// TIA Portal V18 export
// export: Created 2026-06-08T06:16:14.4955932Z, ExportSetting WithDefaults, DisplayName Totally Integrated Automation Portal, DisplayVersion V18, DisplayName TIA Portal Openness, DisplayVersion V18, DisplayName TIA Portal Version Control Interface, DisplayVersion V18, DisplayName STEP 7 Professional, DisplayVersion V18, DisplayName STEP 7 Safety, DisplayVersion V18, DisplayName WinCC Professional, DisplayVersion V18
FUNCTION "FC_Bon_Chua_Loc" : Void   // FC30, LAD
{ S7_Optimized_Access := 'TRUE' }
VERSION : 0.1
// stored: AutoNumber true, IsIECCheckEnabled false, SetENOAutomatically false, UDAEnableTagReadback false
BEGIN

REGION Network 1: Gated HMI AI_LSH3310_Pheu_Cao qua Sim Mode
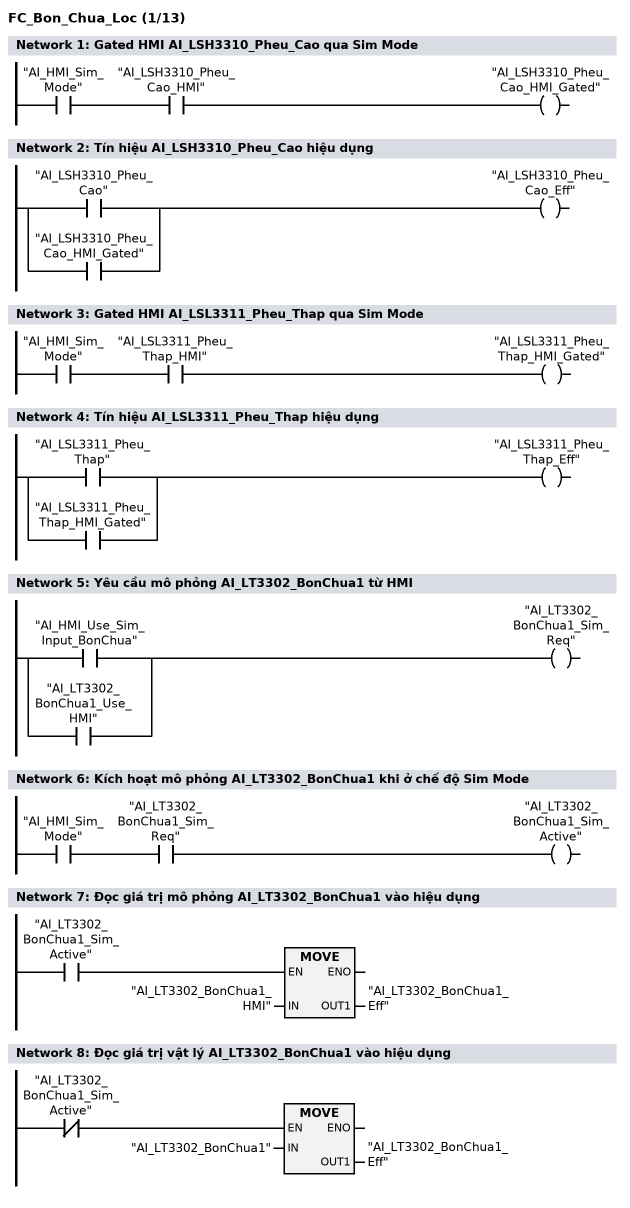
   RUNG wire#powerrail
      Contact( "AI_HMI_Sim_Mode" )
      Contact( "AI_LSH3310_Pheu_Cao_HMI" )
      Coil( "AI_LSH3310_Pheu_Cao_HMI_Gated" )
   END_RUNG
   // the same network as SCL:
   "AI_LSH3310_Pheu_Cao_HMI_Gated" := "AI_HMI_Sim_Mode" AND "AI_LSH3310_Pheu_Cao_HMI";
END_REGION

REGION Network 2: Tín hiệu AI_LSH3310_Pheu_Cao hiệu dụng
   RUNG wire#powerrail
      Contact( "AI_LSH3310_Pheu_Cao" )
      wire#w1
      Coil( "AI_LSH3310_Pheu_Cao_Eff" )
   END_RUNG
   RUNG wire#powerrail
      Contact( "AI_LSH3310_Pheu_Cao_HMI_Gated" )
   END_RUNG wire#w1
   // the same network as SCL:
   "AI_LSH3310_Pheu_Cao_Eff" := "AI_LSH3310_Pheu_Cao" OR "AI_LSH3310_Pheu_Cao_HMI_Gated";
END_REGION

REGION Network 3: Gated HMI AI_LSL3311_Pheu_Thap qua Sim Mode
   RUNG wire#powerrail
      Contact( "AI_HMI_Sim_Mode" )
      Contact( "AI_LSL3311_Pheu_Thap_HMI" )
      Coil( "AI_LSL3311_Pheu_Thap_HMI_Gated" )
   END_RUNG
   // the same network as SCL:
   "AI_LSL3311_Pheu_Thap_HMI_Gated" := "AI_HMI_Sim_Mode" AND "AI_LSL3311_Pheu_Thap_HMI";
END_REGION

REGION Network 4: Tín hiệu AI_LSL3311_Pheu_Thap hiệu dụng
   RUNG wire#powerrail
      Contact( "AI_LSL3311_Pheu_Thap" )
      wire#w1
      Coil( "AI_LSL3311_Pheu_Thap_Eff" )
   END_RUNG
   RUNG wire#powerrail
      Contact( "AI_LSL3311_Pheu_Thap_HMI_Gated" )
   END_RUNG wire#w1
   // the same network as SCL:
   "AI_LSL3311_Pheu_Thap_Eff" := "AI_LSL3311_Pheu_Thap" OR "AI_LSL3311_Pheu_Thap_HMI_Gated";
END_REGION

REGION Network 5: Yêu cầu mô phỏng AI_LT3302_BonChua1 từ HMI
   RUNG wire#powerrail
      Contact( "AI_HMI_Use_Sim_Input_BonChua" )
      wire#w1
      Coil( "AI_LT3302_BonChua1_Sim_Req" )
   END_RUNG
   RUNG wire#powerrail
      Contact( "AI_LT3302_BonChua1_Use_HMI" )
   END_RUNG wire#w1
   // the same network as SCL:
   "AI_LT3302_BonChua1_Sim_Req" := "AI_HMI_Use_Sim_Input_BonChua" OR "AI_LT3302_BonChua1_Use_HMI";
END_REGION

REGION Network 6: Kích hoạt mô phỏng AI_LT3302_BonChua1 khi ở chế độ Sim Mode
   RUNG wire#powerrail
      Contact( "AI_HMI_Sim_Mode" )
      Contact( "AI_LT3302_BonChua1_Sim_Req" )
      Coil( "AI_LT3302_BonChua1_Sim_Active" )
   END_RUNG
   // the same network as SCL:
   "AI_LT3302_BonChua1_Sim_Active" := "AI_HMI_Sim_Mode" AND "AI_LT3302_BonChua1_Sim_Req";
END_REGION

REGION Network 7: Đọc giá trị mô phỏng AI_LT3302_BonChua1 vào hiệu dụng
   RUNG wire#powerrail
      Contact( "AI_LT3302_BonChua1_Sim_Active" )
      { S7_GenerateENO := "TRUE" } Move(in := "AI_LT3302_BonChua1_HMI", out1 => "AI_LT3302_BonChua1_Eff")
   END_RUNG
   // the same network as SCL:
   IF "AI_LT3302_BonChua1_Sim_Active" THEN "AI_LT3302_BonChua1_Eff" := "AI_LT3302_BonChua1_HMI"; END_IF;
END_REGION

REGION Network 8: Đọc giá trị vật lý AI_LT3302_BonChua1 vào hiệu dụng
   RUNG wire#powerrail
      I_Contact( "AI_LT3302_BonChua1_Sim_Active" )
      { S7_GenerateENO := "TRUE" } Move(in := "AI_LT3302_BonChua1", out1 => "AI_LT3302_BonChua1_Eff")
   END_RUNG
   // the same network as SCL:
   IF NOT "AI_LT3302_BonChua1_Sim_Active" THEN "AI_LT3302_BonChua1_Eff" := "AI_LT3302_BonChua1"; END_IF;
END_REGION

REGION Network 9: Yêu cầu mô phỏng AI_TT3301_BonChua1 từ HMI
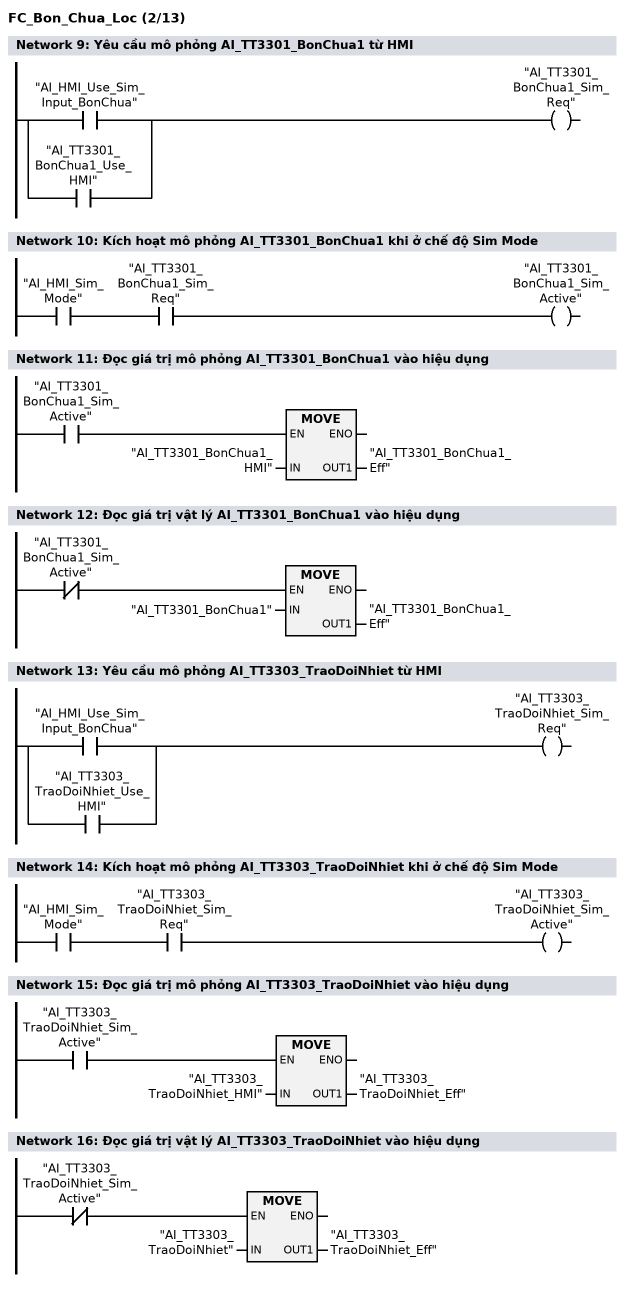
   RUNG wire#powerrail
      Contact( "AI_HMI_Use_Sim_Input_BonChua" )
      wire#w1
      Coil( "AI_TT3301_BonChua1_Sim_Req" )
   END_RUNG
   RUNG wire#powerrail
      Contact( "AI_TT3301_BonChua1_Use_HMI" )
   END_RUNG wire#w1
   // the same network as SCL:
   "AI_TT3301_BonChua1_Sim_Req" := "AI_HMI_Use_Sim_Input_BonChua" OR "AI_TT3301_BonChua1_Use_HMI";
END_REGION

REGION Network 10: Kích hoạt mô phỏng AI_TT3301_BonChua1 khi ở chế độ Sim Mode
   RUNG wire#powerrail
      Contact( "AI_HMI_Sim_Mode" )
      Contact( "AI_TT3301_BonChua1_Sim_Req" )
      Coil( "AI_TT3301_BonChua1_Sim_Active" )
   END_RUNG
   // the same network as SCL:
   "AI_TT3301_BonChua1_Sim_Active" := "AI_HMI_Sim_Mode" AND "AI_TT3301_BonChua1_Sim_Req";
END_REGION

REGION Network 11: Đọc giá trị mô phỏng AI_TT3301_BonChua1 vào hiệu dụng
   RUNG wire#powerrail
      Contact( "AI_TT3301_BonChua1_Sim_Active" )
      { S7_GenerateENO := "TRUE" } Move(in := "AI_TT3301_BonChua1_HMI", out1 => "AI_TT3301_BonChua1_Eff")
   END_RUNG
   // the same network as SCL:
   IF "AI_TT3301_BonChua1_Sim_Active" THEN "AI_TT3301_BonChua1_Eff" := "AI_TT3301_BonChua1_HMI"; END_IF;
END_REGION

REGION Network 12: Đọc giá trị vật lý AI_TT3301_BonChua1 vào hiệu dụng
   RUNG wire#powerrail
      I_Contact( "AI_TT3301_BonChua1_Sim_Active" )
      { S7_GenerateENO := "TRUE" } Move(in := "AI_TT3301_BonChua1", out1 => "AI_TT3301_BonChua1_Eff")
   END_RUNG
   // the same network as SCL:
   IF NOT "AI_TT3301_BonChua1_Sim_Active" THEN "AI_TT3301_BonChua1_Eff" := "AI_TT3301_BonChua1"; END_IF;
END_REGION

REGION Network 13: Yêu cầu mô phỏng AI_TT3303_TraoDoiNhiet từ HMI
   RUNG wire#powerrail
      Contact( "AI_HMI_Use_Sim_Input_BonChua" )
      wire#w1
      Coil( "AI_TT3303_TraoDoiNhiet_Sim_Req" )
   END_RUNG
   RUNG wire#powerrail
      Contact( "AI_TT3303_TraoDoiNhiet_Use_HMI" )
   END_RUNG wire#w1
   // the same network as SCL:
   "AI_TT3303_TraoDoiNhiet_Sim_Req" := "AI_HMI_Use_Sim_Input_BonChua" OR "AI_TT3303_TraoDoiNhiet_Use_HMI";
END_REGION

REGION Network 14: Kích hoạt mô phỏng AI_TT3303_TraoDoiNhiet khi ở chế độ Sim Mode
   RUNG wire#powerrail
      Contact( "AI_HMI_Sim_Mode" )
      Contact( "AI_TT3303_TraoDoiNhiet_Sim_Req" )
      Coil( "AI_TT3303_TraoDoiNhiet_Sim_Active" )
   END_RUNG
   // the same network as SCL:
   "AI_TT3303_TraoDoiNhiet_Sim_Active" := "AI_HMI_Sim_Mode" AND "AI_TT3303_TraoDoiNhiet_Sim_Req";
END_REGION

REGION Network 15: Đọc giá trị mô phỏng AI_TT3303_TraoDoiNhiet vào hiệu dụng
   RUNG wire#powerrail
      Contact( "AI_TT3303_TraoDoiNhiet_Sim_Active" )
      { S7_GenerateENO := "TRUE" } Move(in := "AI_TT3303_TraoDoiNhiet_HMI", out1 => "AI_TT3303_TraoDoiNhiet_Eff")
   END_RUNG
   // the same network as SCL:
   IF "AI_TT3303_TraoDoiNhiet_Sim_Active" THEN
       "AI_TT3303_TraoDoiNhiet_Eff" := "AI_TT3303_TraoDoiNhiet_HMI";
   END_IF;
END_REGION

REGION Network 16: Đọc giá trị vật lý AI_TT3303_TraoDoiNhiet vào hiệu dụng
   RUNG wire#powerrail
      I_Contact( "AI_TT3303_TraoDoiNhiet_Sim_Active" )
      { S7_GenerateENO := "TRUE" } Move(in := "AI_TT3303_TraoDoiNhiet", out1 => "AI_TT3303_TraoDoiNhiet_Eff")
   END_RUNG
   // the same network as SCL:
   IF NOT "AI_TT3303_TraoDoiNhiet_Sim_Active" THEN
       "AI_TT3303_TraoDoiNhiet_Eff" := "AI_TT3303_TraoDoiNhiet";
   END_IF;
END_REGION

REGION Network 17: Yêu cầu mô phỏng AI_LT3307_BonChua2 từ HMI
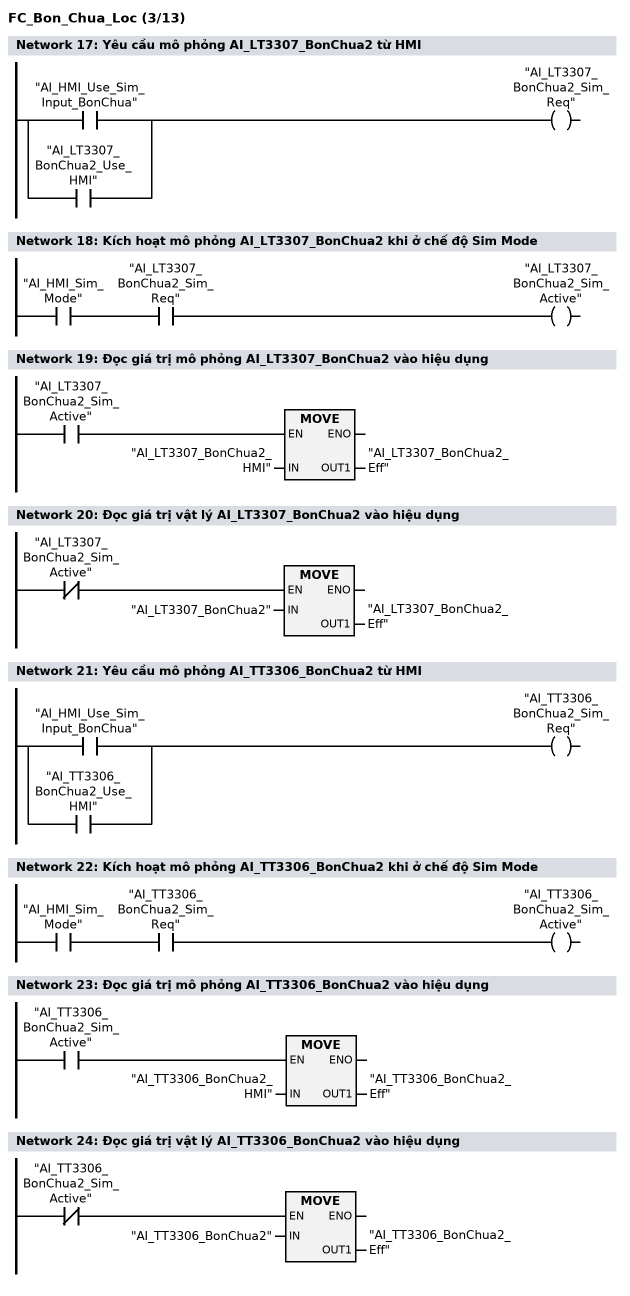
   RUNG wire#powerrail
      Contact( "AI_HMI_Use_Sim_Input_BonChua" )
      wire#w1
      Coil( "AI_LT3307_BonChua2_Sim_Req" )
   END_RUNG
   RUNG wire#powerrail
      Contact( "AI_LT3307_BonChua2_Use_HMI" )
   END_RUNG wire#w1
   // the same network as SCL:
   "AI_LT3307_BonChua2_Sim_Req" := "AI_HMI_Use_Sim_Input_BonChua" OR "AI_LT3307_BonChua2_Use_HMI";
END_REGION

REGION Network 18: Kích hoạt mô phỏng AI_LT3307_BonChua2 khi ở chế độ Sim Mode
   RUNG wire#powerrail
      Contact( "AI_HMI_Sim_Mode" )
      Contact( "AI_LT3307_BonChua2_Sim_Req" )
      Coil( "AI_LT3307_BonChua2_Sim_Active" )
   END_RUNG
   // the same network as SCL:
   "AI_LT3307_BonChua2_Sim_Active" := "AI_HMI_Sim_Mode" AND "AI_LT3307_BonChua2_Sim_Req";
END_REGION

REGION Network 19: Đọc giá trị mô phỏng AI_LT3307_BonChua2 vào hiệu dụng
   RUNG wire#powerrail
      Contact( "AI_LT3307_BonChua2_Sim_Active" )
      { S7_GenerateENO := "TRUE" } Move(in := "AI_LT3307_BonChua2_HMI", out1 => "AI_LT3307_BonChua2_Eff")
   END_RUNG
   // the same network as SCL:
   IF "AI_LT3307_BonChua2_Sim_Active" THEN "AI_LT3307_BonChua2_Eff" := "AI_LT3307_BonChua2_HMI"; END_IF;
END_REGION

REGION Network 20: Đọc giá trị vật lý AI_LT3307_BonChua2 vào hiệu dụng
   RUNG wire#powerrail
      I_Contact( "AI_LT3307_BonChua2_Sim_Active" )
      { S7_GenerateENO := "TRUE" } Move(in := "AI_LT3307_BonChua2", out1 => "AI_LT3307_BonChua2_Eff")
   END_RUNG
   // the same network as SCL:
   IF NOT "AI_LT3307_BonChua2_Sim_Active" THEN "AI_LT3307_BonChua2_Eff" := "AI_LT3307_BonChua2"; END_IF;
END_REGION

REGION Network 21: Yêu cầu mô phỏng AI_TT3306_BonChua2 từ HMI
   RUNG wire#powerrail
      Contact( "AI_HMI_Use_Sim_Input_BonChua" )
      wire#w1
      Coil( "AI_TT3306_BonChua2_Sim_Req" )
   END_RUNG
   RUNG wire#powerrail
      Contact( "AI_TT3306_BonChua2_Use_HMI" )
   END_RUNG wire#w1
   // the same network as SCL:
   "AI_TT3306_BonChua2_Sim_Req" := "AI_HMI_Use_Sim_Input_BonChua" OR "AI_TT3306_BonChua2_Use_HMI";
END_REGION

REGION Network 22: Kích hoạt mô phỏng AI_TT3306_BonChua2 khi ở chế độ Sim Mode
   RUNG wire#powerrail
      Contact( "AI_HMI_Sim_Mode" )
      Contact( "AI_TT3306_BonChua2_Sim_Req" )
      Coil( "AI_TT3306_BonChua2_Sim_Active" )
   END_RUNG
   // the same network as SCL:
   "AI_TT3306_BonChua2_Sim_Active" := "AI_HMI_Sim_Mode" AND "AI_TT3306_BonChua2_Sim_Req";
END_REGION

REGION Network 23: Đọc giá trị mô phỏng AI_TT3306_BonChua2 vào hiệu dụng
   RUNG wire#powerrail
      Contact( "AI_TT3306_BonChua2_Sim_Active" )
      { S7_GenerateENO := "TRUE" } Move(in := "AI_TT3306_BonChua2_HMI", out1 => "AI_TT3306_BonChua2_Eff")
   END_RUNG
   // the same network as SCL:
   IF "AI_TT3306_BonChua2_Sim_Active" THEN "AI_TT3306_BonChua2_Eff" := "AI_TT3306_BonChua2_HMI"; END_IF;
END_REGION

REGION Network 24: Đọc giá trị vật lý AI_TT3306_BonChua2 vào hiệu dụng
   RUNG wire#powerrail
      I_Contact( "AI_TT3306_BonChua2_Sim_Active" )
      { S7_GenerateENO := "TRUE" } Move(in := "AI_TT3306_BonChua2", out1 => "AI_TT3306_BonChua2_Eff")
   END_RUNG
   // the same network as SCL:
   IF NOT "AI_TT3306_BonChua2_Sim_Active" THEN "AI_TT3306_BonChua2_Eff" := "AI_TT3306_BonChua2"; END_IF;
END_REGION

REGION Network 25: Yêu cầu mô phỏng AI_PI3308_Truoc_Filter từ HMI
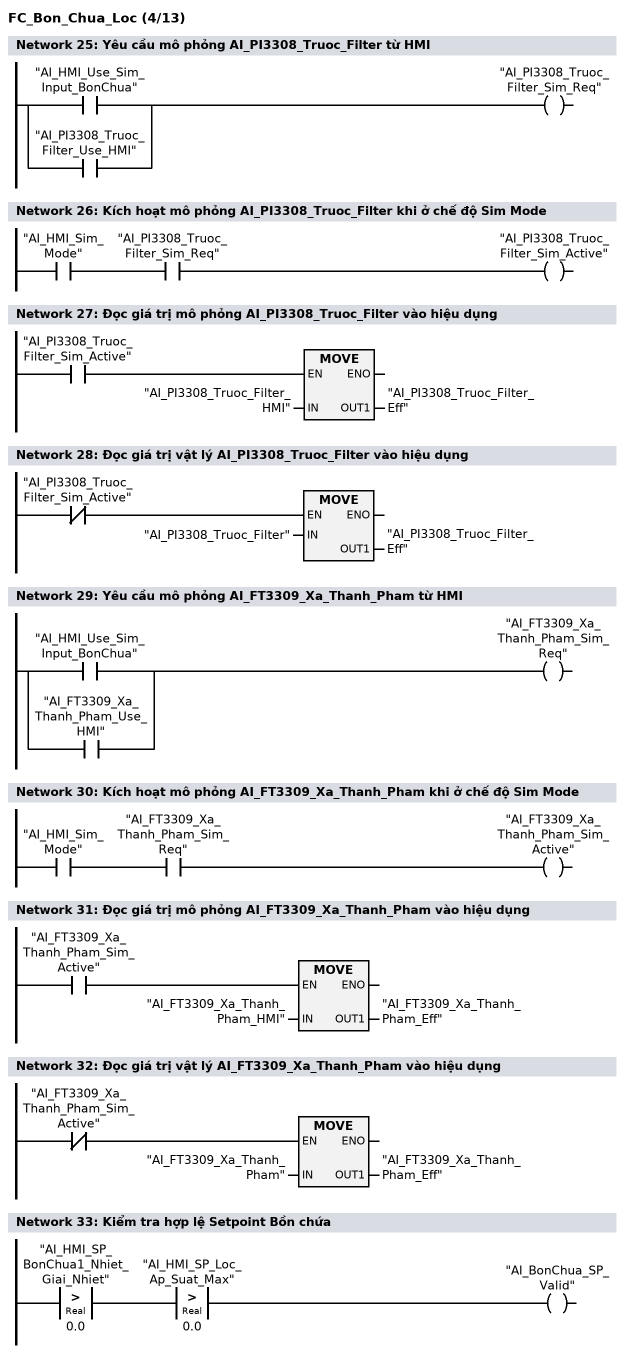
   RUNG wire#powerrail
      Contact( "AI_HMI_Use_Sim_Input_BonChua" )
      wire#w1
      Coil( "AI_PI3308_Truoc_Filter_Sim_Req" )
   END_RUNG
   RUNG wire#powerrail
      Contact( "AI_PI3308_Truoc_Filter_Use_HMI" )
   END_RUNG wire#w1
   // the same network as SCL:
   "AI_PI3308_Truoc_Filter_Sim_Req" := "AI_HMI_Use_Sim_Input_BonChua" OR "AI_PI3308_Truoc_Filter_Use_HMI";
END_REGION

REGION Network 26: Kích hoạt mô phỏng AI_PI3308_Truoc_Filter khi ở chế độ Sim Mode
   RUNG wire#powerrail
      Contact( "AI_HMI_Sim_Mode" )
      Contact( "AI_PI3308_Truoc_Filter_Sim_Req" )
      Coil( "AI_PI3308_Truoc_Filter_Sim_Active" )
   END_RUNG
   // the same network as SCL:
   "AI_PI3308_Truoc_Filter_Sim_Active" := "AI_HMI_Sim_Mode" AND "AI_PI3308_Truoc_Filter_Sim_Req";
END_REGION

REGION Network 27: Đọc giá trị mô phỏng AI_PI3308_Truoc_Filter vào hiệu dụng
   RUNG wire#powerrail
      Contact( "AI_PI3308_Truoc_Filter_Sim_Active" )
      { S7_GenerateENO := "TRUE" } Move(in := "AI_PI3308_Truoc_Filter_HMI", out1 => "AI_PI3308_Truoc_Filter_Eff")
   END_RUNG
   // the same network as SCL:
   IF "AI_PI3308_Truoc_Filter_Sim_Active" THEN
       "AI_PI3308_Truoc_Filter_Eff" := "AI_PI3308_Truoc_Filter_HMI";
   END_IF;
END_REGION

REGION Network 28: Đọc giá trị vật lý AI_PI3308_Truoc_Filter vào hiệu dụng
   RUNG wire#powerrail
      I_Contact( "AI_PI3308_Truoc_Filter_Sim_Active" )
      { S7_GenerateENO := "TRUE" } Move(in := "AI_PI3308_Truoc_Filter", out1 => "AI_PI3308_Truoc_Filter_Eff")
   END_RUNG
   // the same network as SCL:
   IF NOT "AI_PI3308_Truoc_Filter_Sim_Active" THEN
       "AI_PI3308_Truoc_Filter_Eff" := "AI_PI3308_Truoc_Filter";
   END_IF;
END_REGION

REGION Network 29: Yêu cầu mô phỏng AI_FT3309_Xa_Thanh_Pham từ HMI
   RUNG wire#powerrail
      Contact( "AI_HMI_Use_Sim_Input_BonChua" )
      wire#w1
      Coil( "AI_FT3309_Xa_Thanh_Pham_Sim_Req" )
   END_RUNG
   RUNG wire#powerrail
      Contact( "AI_FT3309_Xa_Thanh_Pham_Use_HMI" )
   END_RUNG wire#w1
   // the same network as SCL:
   "AI_FT3309_Xa_Thanh_Pham_Sim_Req" := "AI_HMI_Use_Sim_Input_BonChua" OR "AI_FT3309_Xa_Thanh_Pham_Use_HMI";
END_REGION

REGION Network 30: Kích hoạt mô phỏng AI_FT3309_Xa_Thanh_Pham khi ở chế độ Sim Mode
   RUNG wire#powerrail
      Contact( "AI_HMI_Sim_Mode" )
      Contact( "AI_FT3309_Xa_Thanh_Pham_Sim_Req" )
      Coil( "AI_FT3309_Xa_Thanh_Pham_Sim_Active" )
   END_RUNG
   // the same network as SCL:
   "AI_FT3309_Xa_Thanh_Pham_Sim_Active" := "AI_HMI_Sim_Mode" AND "AI_FT3309_Xa_Thanh_Pham_Sim_Req";
END_REGION

REGION Network 31: Đọc giá trị mô phỏng AI_FT3309_Xa_Thanh_Pham vào hiệu dụng
   RUNG wire#powerrail
      Contact( "AI_FT3309_Xa_Thanh_Pham_Sim_Active" )
      { S7_GenerateENO := "TRUE" } Move(in := "AI_FT3309_Xa_Thanh_Pham_HMI", out1 => "AI_FT3309_Xa_Thanh_Pham_Eff")
   END_RUNG
   // the same network as SCL:
   IF "AI_FT3309_Xa_Thanh_Pham_Sim_Active" THEN
       "AI_FT3309_Xa_Thanh_Pham_Eff" := "AI_FT3309_Xa_Thanh_Pham_HMI";
   END_IF;
END_REGION

REGION Network 32: Đọc giá trị vật lý AI_FT3309_Xa_Thanh_Pham vào hiệu dụng
   RUNG wire#powerrail
      I_Contact( "AI_FT3309_Xa_Thanh_Pham_Sim_Active" )
      { S7_GenerateENO := "TRUE" } Move(in := "AI_FT3309_Xa_Thanh_Pham", out1 => "AI_FT3309_Xa_Thanh_Pham_Eff")
   END_RUNG
   // the same network as SCL:
   IF NOT "AI_FT3309_Xa_Thanh_Pham_Sim_Active" THEN
       "AI_FT3309_Xa_Thanh_Pham_Eff" := "AI_FT3309_Xa_Thanh_Pham";
   END_IF;
END_REGION

REGION Network 33: Kiểm tra hợp lệ Setpoint Bồn chứa
   RUNG wire#powerrail
      { S7_Templates := "SrcType := Real" } GT_Contact(in1 := "AI_HMI_SP_BonChua1_Nhiet_Giai_Nhiet", in2 := 0.0)
      { S7_Templates := "SrcType := Real" } GT_Contact(in1 := "AI_HMI_SP_Loc_Ap_Suat_Max", in2 := 0.0)
      Coil( "AI_BonChua_SP_Valid" )
   END_RUNG
   // the same network as SCL:
   "AI_BonChua_SP_Valid" := ("AI_HMI_SP_BonChua1_Nhiet_Giai_Nhiet" > 0.0) AND ("AI_HMI_SP_Loc_Ap_Suat_Max" > 0.0);
END_REGION

REGION Network 34: Stop Storage - reset AI_BonChua_Step_Nhan_Dich
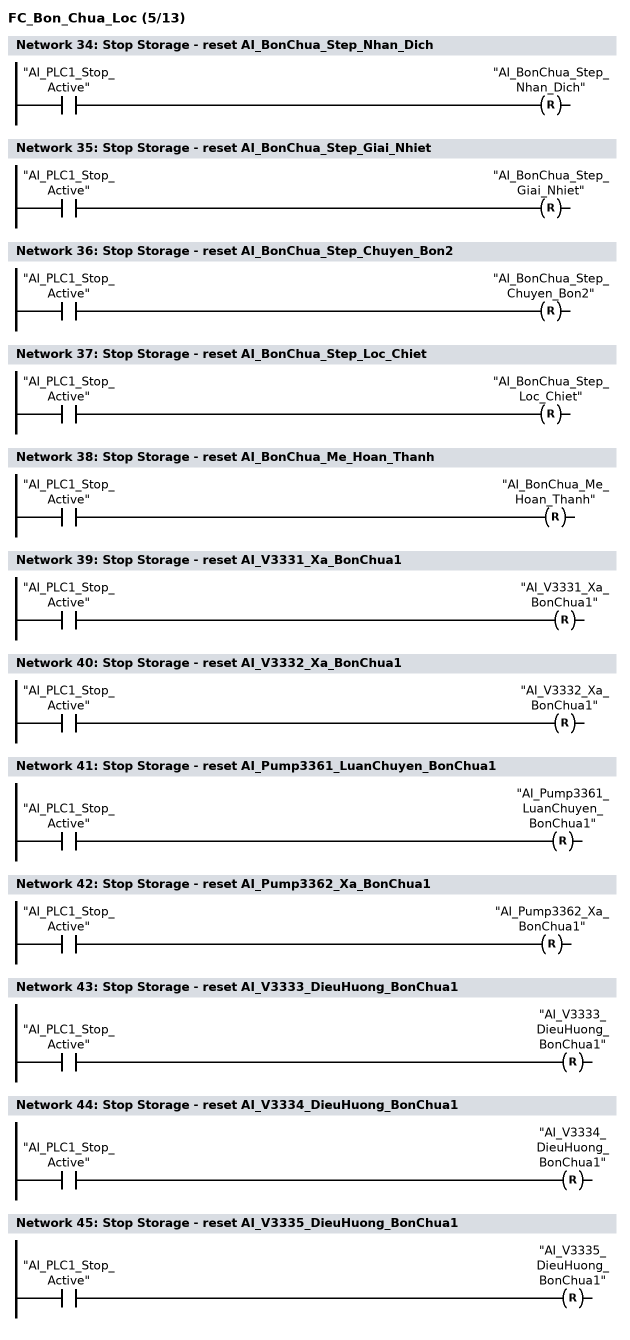
   RUNG wire#powerrail
      Contact( "AI_PLC1_Stop_Active" )
      R_Coil( "AI_BonChua_Step_Nhan_Dich" )
   END_RUNG
   // the same network as SCL:
   IF "AI_PLC1_Stop_Active" THEN "AI_BonChua_Step_Nhan_Dich" := FALSE; END_IF;
END_REGION

REGION Network 35: Stop Storage - reset AI_BonChua_Step_Giai_Nhiet
   RUNG wire#powerrail
      Contact( "AI_PLC1_Stop_Active" )
      R_Coil( "AI_BonChua_Step_Giai_Nhiet" )
   END_RUNG
   // the same network as SCL:
   IF "AI_PLC1_Stop_Active" THEN "AI_BonChua_Step_Giai_Nhiet" := FALSE; END_IF;
END_REGION

REGION Network 36: Stop Storage - reset AI_BonChua_Step_Chuyen_Bon2
   RUNG wire#powerrail
      Contact( "AI_PLC1_Stop_Active" )
      R_Coil( "AI_BonChua_Step_Chuyen_Bon2" )
   END_RUNG
   // the same network as SCL:
   IF "AI_PLC1_Stop_Active" THEN "AI_BonChua_Step_Chuyen_Bon2" := FALSE; END_IF;
END_REGION

REGION Network 37: Stop Storage - reset AI_BonChua_Step_Loc_Chiet
   RUNG wire#powerrail
      Contact( "AI_PLC1_Stop_Active" )
      R_Coil( "AI_BonChua_Step_Loc_Chiet" )
   END_RUNG
   // the same network as SCL:
   IF "AI_PLC1_Stop_Active" THEN "AI_BonChua_Step_Loc_Chiet" := FALSE; END_IF;
END_REGION

REGION Network 38: Stop Storage - reset AI_BonChua_Me_Hoan_Thanh
   RUNG wire#powerrail
      Contact( "AI_PLC1_Stop_Active" )
      R_Coil( "AI_BonChua_Me_Hoan_Thanh" )
   END_RUNG
   // the same network as SCL:
   IF "AI_PLC1_Stop_Active" THEN "AI_BonChua_Me_Hoan_Thanh" := FALSE; END_IF;
END_REGION

REGION Network 39: Stop Storage - reset AI_V3331_Xa_BonChua1
   RUNG wire#powerrail
      Contact( "AI_PLC1_Stop_Active" )
      R_Coil( "AI_V3331_Xa_BonChua1" )
   END_RUNG
   // the same network as SCL:
   IF "AI_PLC1_Stop_Active" THEN "AI_V3331_Xa_BonChua1" := FALSE; END_IF;
END_REGION

REGION Network 40: Stop Storage - reset AI_V3332_Xa_BonChua1
   RUNG wire#powerrail
      Contact( "AI_PLC1_Stop_Active" )
      R_Coil( "AI_V3332_Xa_BonChua1" )
   END_RUNG
   // the same network as SCL:
   IF "AI_PLC1_Stop_Active" THEN "AI_V3332_Xa_BonChua1" := FALSE; END_IF;
END_REGION

REGION Network 41: Stop Storage - reset AI_Pump3361_LuanChuyen_BonChua1
   RUNG wire#powerrail
      Contact( "AI_PLC1_Stop_Active" )
      R_Coil( "AI_Pump3361_LuanChuyen_BonChua1" )
   END_RUNG
   // the same network as SCL:
   IF "AI_PLC1_Stop_Active" THEN "AI_Pump3361_LuanChuyen_BonChua1" := FALSE; END_IF;
END_REGION

REGION Network 42: Stop Storage - reset AI_Pump3362_Xa_BonChua1
   RUNG wire#powerrail
      Contact( "AI_PLC1_Stop_Active" )
      R_Coil( "AI_Pump3362_Xa_BonChua1" )
   END_RUNG
   // the same network as SCL:
   IF "AI_PLC1_Stop_Active" THEN "AI_Pump3362_Xa_BonChua1" := FALSE; END_IF;
END_REGION

REGION Network 43: Stop Storage - reset AI_V3333_DieuHuong_BonChua1
   RUNG wire#powerrail
      Contact( "AI_PLC1_Stop_Active" )
      R_Coil( "AI_V3333_DieuHuong_BonChua1" )
   END_RUNG
   // the same network as SCL:
   IF "AI_PLC1_Stop_Active" THEN "AI_V3333_DieuHuong_BonChua1" := FALSE; END_IF;
END_REGION

REGION Network 44: Stop Storage - reset AI_V3334_DieuHuong_BonChua1
   RUNG wire#powerrail
      Contact( "AI_PLC1_Stop_Active" )
      R_Coil( "AI_V3334_DieuHuong_BonChua1" )
   END_RUNG
   // the same network as SCL:
   IF "AI_PLC1_Stop_Active" THEN "AI_V3334_DieuHuong_BonChua1" := FALSE; END_IF;
END_REGION

REGION Network 45: Stop Storage - reset AI_V3335_DieuHuong_BonChua1
   RUNG wire#powerrail
      Contact( "AI_PLC1_Stop_Active" )
      R_Coil( "AI_V3335_DieuHuong_BonChua1" )
   END_RUNG
   // the same network as SCL:
   IF "AI_PLC1_Stop_Active" THEN "AI_V3335_DieuHuong_BonChua1" := FALSE; END_IF;
END_REGION

REGION Network 46: Stop Storage - reset AI_V3338_Xa_BonChua2
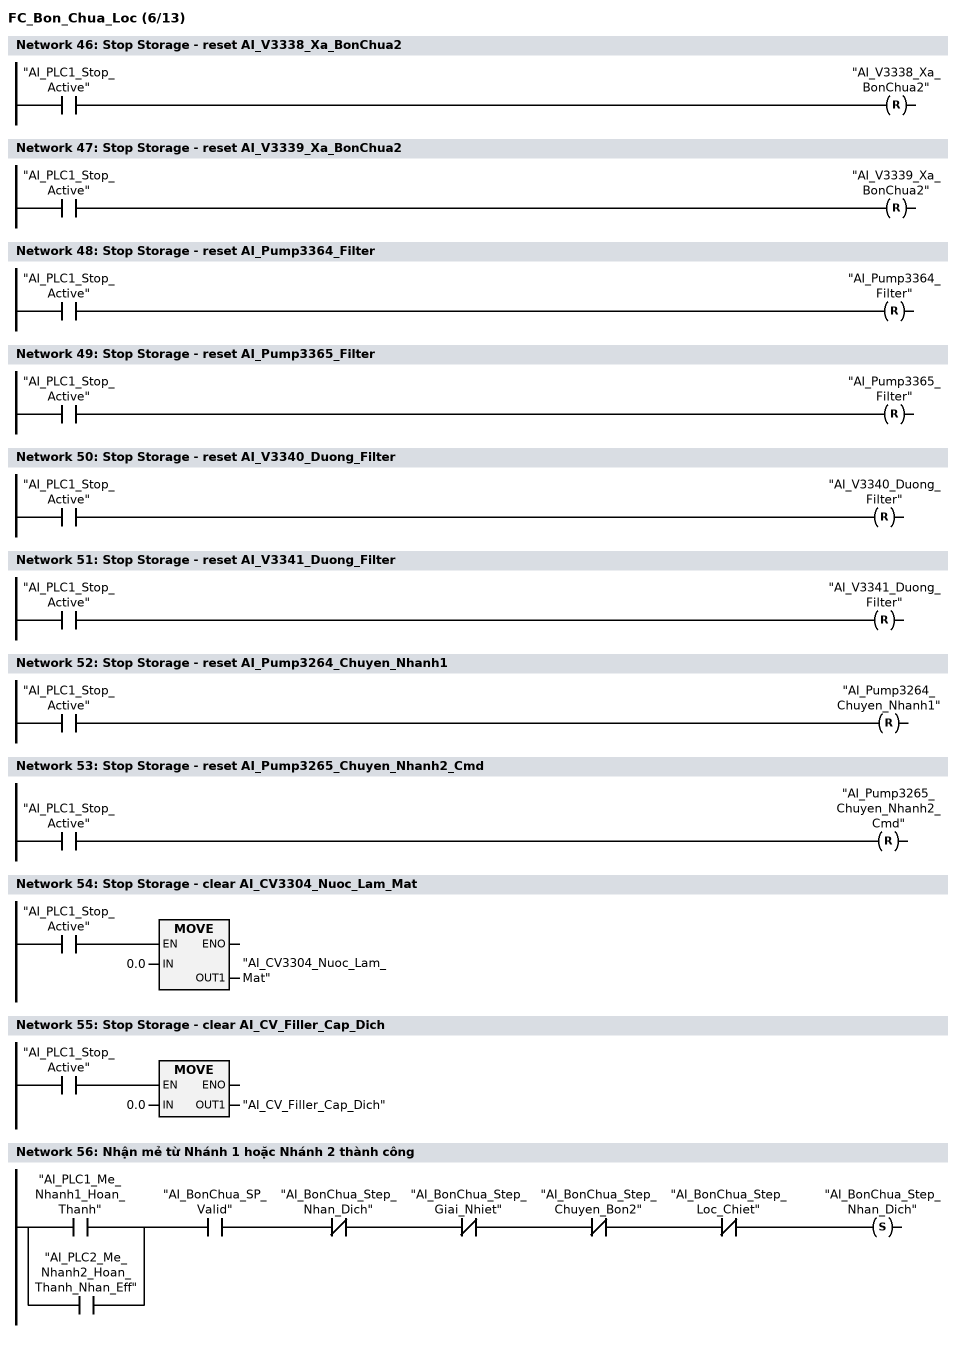
   RUNG wire#powerrail
      Contact( "AI_PLC1_Stop_Active" )
      R_Coil( "AI_V3338_Xa_BonChua2" )
   END_RUNG
   // the same network as SCL:
   IF "AI_PLC1_Stop_Active" THEN "AI_V3338_Xa_BonChua2" := FALSE; END_IF;
END_REGION

REGION Network 47: Stop Storage - reset AI_V3339_Xa_BonChua2
   RUNG wire#powerrail
      Contact( "AI_PLC1_Stop_Active" )
      R_Coil( "AI_V3339_Xa_BonChua2" )
   END_RUNG
   // the same network as SCL:
   IF "AI_PLC1_Stop_Active" THEN "AI_V3339_Xa_BonChua2" := FALSE; END_IF;
END_REGION

REGION Network 48: Stop Storage - reset AI_Pump3364_Filter
   RUNG wire#powerrail
      Contact( "AI_PLC1_Stop_Active" )
      R_Coil( "AI_Pump3364_Filter" )
   END_RUNG
   // the same network as SCL:
   IF "AI_PLC1_Stop_Active" THEN "AI_Pump3364_Filter" := FALSE; END_IF;
END_REGION

REGION Network 49: Stop Storage - reset AI_Pump3365_Filter
   RUNG wire#powerrail
      Contact( "AI_PLC1_Stop_Active" )
      R_Coil( "AI_Pump3365_Filter" )
   END_RUNG
   // the same network as SCL:
   IF "AI_PLC1_Stop_Active" THEN "AI_Pump3365_Filter" := FALSE; END_IF;
END_REGION

REGION Network 50: Stop Storage - reset AI_V3340_Duong_Filter
   RUNG wire#powerrail
      Contact( "AI_PLC1_Stop_Active" )
      R_Coil( "AI_V3340_Duong_Filter" )
   END_RUNG
   // the same network as SCL:
   IF "AI_PLC1_Stop_Active" THEN "AI_V3340_Duong_Filter" := FALSE; END_IF;
END_REGION

REGION Network 51: Stop Storage - reset AI_V3341_Duong_Filter
   RUNG wire#powerrail
      Contact( "AI_PLC1_Stop_Active" )
      R_Coil( "AI_V3341_Duong_Filter" )
   END_RUNG
   // the same network as SCL:
   IF "AI_PLC1_Stop_Active" THEN "AI_V3341_Duong_Filter" := FALSE; END_IF;
END_REGION

REGION Network 52: Stop Storage - reset AI_Pump3264_Chuyen_Nhanh1
   RUNG wire#powerrail
      Contact( "AI_PLC1_Stop_Active" )
      R_Coil( "AI_Pump3264_Chuyen_Nhanh1" )
   END_RUNG
   // the same network as SCL:
   IF "AI_PLC1_Stop_Active" THEN "AI_Pump3264_Chuyen_Nhanh1" := FALSE; END_IF;
END_REGION

REGION Network 53: Stop Storage - reset AI_Pump3265_Chuyen_Nhanh2_Cmd
   RUNG wire#powerrail
      Contact( "AI_PLC1_Stop_Active" )
      R_Coil( "AI_Pump3265_Chuyen_Nhanh2_Cmd" )
   END_RUNG
   // the same network as SCL:
   IF "AI_PLC1_Stop_Active" THEN "AI_Pump3265_Chuyen_Nhanh2_Cmd" := FALSE; END_IF;
END_REGION

REGION Network 54: Stop Storage - clear AI_CV3304_Nuoc_Lam_Mat
   RUNG wire#powerrail
      Contact( "AI_PLC1_Stop_Active" )
      { S7_GenerateENO := "TRUE" } Move(in := 0.0, out1 => "AI_CV3304_Nuoc_Lam_Mat")
   END_RUNG
   // the same network as SCL:
   IF "AI_PLC1_Stop_Active" THEN "AI_CV3304_Nuoc_Lam_Mat" := 0.0; END_IF;
END_REGION

REGION Network 55: Stop Storage - clear AI_CV_Filler_Cap_Dich
   RUNG wire#powerrail
      Contact( "AI_PLC1_Stop_Active" )
      { S7_GenerateENO := "TRUE" } Move(in := 0.0, out1 => "AI_CV_Filler_Cap_Dich")
   END_RUNG
   // the same network as SCL:
   IF "AI_PLC1_Stop_Active" THEN "AI_CV_Filler_Cap_Dich" := 0.0; END_IF;
END_REGION

REGION Network 56: Nhận mẻ từ Nhánh 1 hoặc Nhánh 2 thành công
   RUNG wire#powerrail
      Contact( "AI_PLC1_Me_Nhanh1_Hoan_Thanh" )
      wire#w1
      Contact( "AI_BonChua_SP_Valid" )
      I_Contact( "AI_BonChua_Step_Nhan_Dich" )
      I_Contact( "AI_BonChua_Step_Giai_Nhiet" )
      I_Contact( "AI_BonChua_Step_Chuyen_Bon2" )
      I_Contact( "AI_BonChua_Step_Loc_Chiet" )
      S_Coil( "AI_BonChua_Step_Nhan_Dich" )
   END_RUNG
   RUNG wire#powerrail
      Contact( "AI_PLC2_Me_Nhanh2_Hoan_Thanh_Nhan_Eff" )
   END_RUNG wire#w1
   // the same network as SCL:
   IF ("AI_PLC1_Me_Nhanh1_Hoan_Thanh" OR "AI_PLC2_Me_Nhanh2_Hoan_Thanh_Nhan_Eff") AND "AI_BonChua_SP_Valid" AND NOT "AI_BonChua_Step_Nhan_Dich" AND NOT "AI_BonChua_Step_Giai_Nhiet" AND NOT "AI_BonChua_Step_Chuyen_Bon2" AND NOT "AI_BonChua_Step_Loc_Chiet" THEN
       "AI_BonChua_Step_Nhan_Dich" := TRUE;
   END_IF;
END_REGION

REGION Network 57: Báo lỗi setpoint bồn chứa khi nhận mẻ
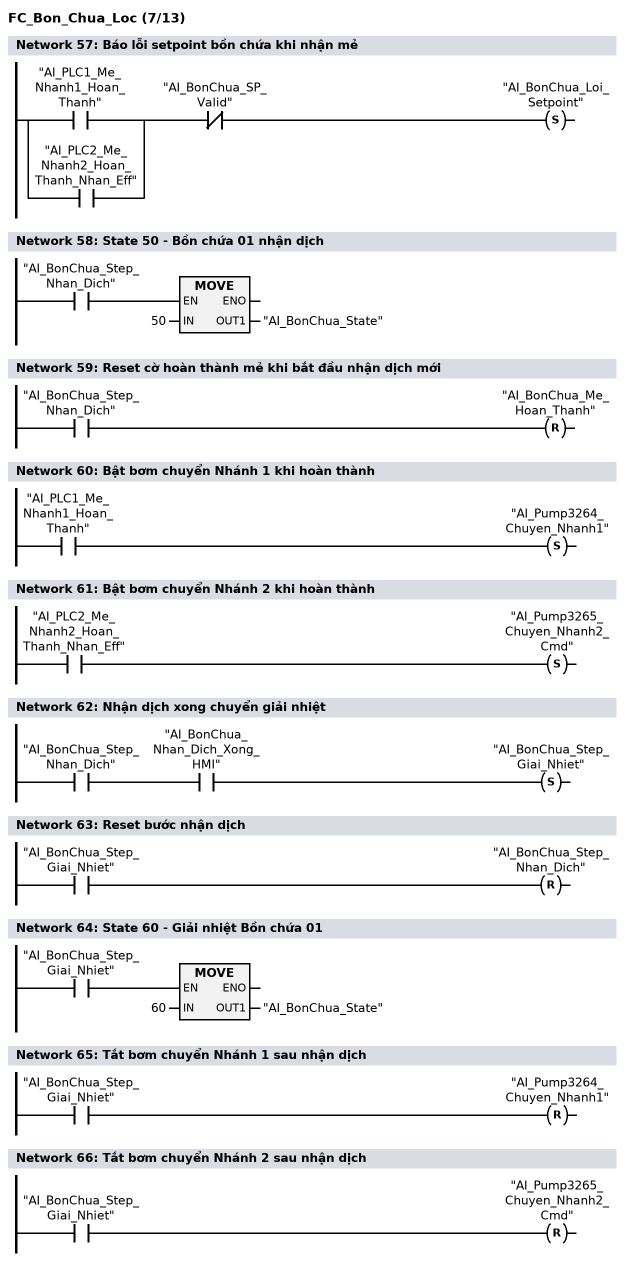
   RUNG wire#powerrail
      Contact( "AI_PLC1_Me_Nhanh1_Hoan_Thanh" )
      wire#w1
      I_Contact( "AI_BonChua_SP_Valid" )
      S_Coil( "AI_BonChua_Loi_Setpoint" )
   END_RUNG
   RUNG wire#powerrail
      Contact( "AI_PLC2_Me_Nhanh2_Hoan_Thanh_Nhan_Eff" )
   END_RUNG wire#w1
   // the same network as SCL:
   IF ("AI_PLC1_Me_Nhanh1_Hoan_Thanh" OR "AI_PLC2_Me_Nhanh2_Hoan_Thanh_Nhan_Eff") AND NOT "AI_BonChua_SP_Valid" THEN
       "AI_BonChua_Loi_Setpoint" := TRUE;
   END_IF;
END_REGION

REGION Network 58: State 50 - Bồn chứa 01 nhận dịch
   RUNG wire#powerrail
      Contact( "AI_BonChua_Step_Nhan_Dich" )
      { S7_GenerateENO := "TRUE" } Move(in := 50, out1 => "AI_BonChua_State")
   END_RUNG
   // the same network as SCL:
   IF "AI_BonChua_Step_Nhan_Dich" THEN "AI_BonChua_State" := 50; END_IF;
END_REGION

REGION Network 59: Reset cờ hoàn thành mẻ khi bắt đầu nhận dịch mới
   RUNG wire#powerrail
      Contact( "AI_BonChua_Step_Nhan_Dich" )
      R_Coil( "AI_BonChua_Me_Hoan_Thanh" )
   END_RUNG
   // the same network as SCL:
   IF "AI_BonChua_Step_Nhan_Dich" THEN "AI_BonChua_Me_Hoan_Thanh" := FALSE; END_IF;
END_REGION

REGION Network 60: Bật bơm chuyển Nhánh 1 khi hoàn thành
   RUNG wire#powerrail
      Contact( "AI_PLC1_Me_Nhanh1_Hoan_Thanh" )
      S_Coil( "AI_Pump3264_Chuyen_Nhanh1" )
   END_RUNG
   // the same network as SCL:
   IF "AI_PLC1_Me_Nhanh1_Hoan_Thanh" THEN "AI_Pump3264_Chuyen_Nhanh1" := TRUE; END_IF;
END_REGION

REGION Network 61: Bật bơm chuyển Nhánh 2 khi hoàn thành
   RUNG wire#powerrail
      Contact( "AI_PLC2_Me_Nhanh2_Hoan_Thanh_Nhan_Eff" )
      S_Coil( "AI_Pump3265_Chuyen_Nhanh2_Cmd" )
   END_RUNG
   // the same network as SCL:
   IF "AI_PLC2_Me_Nhanh2_Hoan_Thanh_Nhan_Eff" THEN "AI_Pump3265_Chuyen_Nhanh2_Cmd" := TRUE; END_IF;
END_REGION

REGION Network 62: Nhận dịch xong chuyển giải nhiệt
   RUNG wire#powerrail
      Contact( "AI_BonChua_Step_Nhan_Dich" )
      Contact( "AI_BonChua_Nhan_Dich_Xong_HMI" )
      S_Coil( "AI_BonChua_Step_Giai_Nhiet" )
   END_RUNG
   // the same network as SCL:
   IF "AI_BonChua_Step_Nhan_Dich" AND "AI_BonChua_Nhan_Dich_Xong_HMI" THEN
       "AI_BonChua_Step_Giai_Nhiet" := TRUE;
   END_IF;
END_REGION

REGION Network 63: Reset bước nhận dịch
   RUNG wire#powerrail
      Contact( "AI_BonChua_Step_Giai_Nhiet" )
      R_Coil( "AI_BonChua_Step_Nhan_Dich" )
   END_RUNG
   // the same network as SCL:
   IF "AI_BonChua_Step_Giai_Nhiet" THEN "AI_BonChua_Step_Nhan_Dich" := FALSE; END_IF;
END_REGION

REGION Network 64: State 60 - Giải nhiệt Bồn chứa 01
   RUNG wire#powerrail
      Contact( "AI_BonChua_Step_Giai_Nhiet" )
      { S7_GenerateENO := "TRUE" } Move(in := 60, out1 => "AI_BonChua_State")
   END_RUNG
   // the same network as SCL:
   IF "AI_BonChua_Step_Giai_Nhiet" THEN "AI_BonChua_State" := 60; END_IF;
END_REGION

REGION Network 65: Tắt bơm chuyển Nhánh 1 sau nhận dịch
   RUNG wire#powerrail
      Contact( "AI_BonChua_Step_Giai_Nhiet" )
      R_Coil( "AI_Pump3264_Chuyen_Nhanh1" )
   END_RUNG
   // the same network as SCL:
   IF "AI_BonChua_Step_Giai_Nhiet" THEN "AI_Pump3264_Chuyen_Nhanh1" := FALSE; END_IF;
END_REGION

REGION Network 66: Tắt bơm chuyển Nhánh 2 sau nhận dịch
   RUNG wire#powerrail
      Contact( "AI_BonChua_Step_Giai_Nhiet" )
      R_Coil( "AI_Pump3265_Chuyen_Nhanh2_Cmd" )
   END_RUNG
   // the same network as SCL:
   IF "AI_BonChua_Step_Giai_Nhiet" THEN "AI_Pump3265_Chuyen_Nhanh2_Cmd" := FALSE; END_IF;
END_REGION

REGION Network 67: Reset cờ hoàn thành Nhánh 1
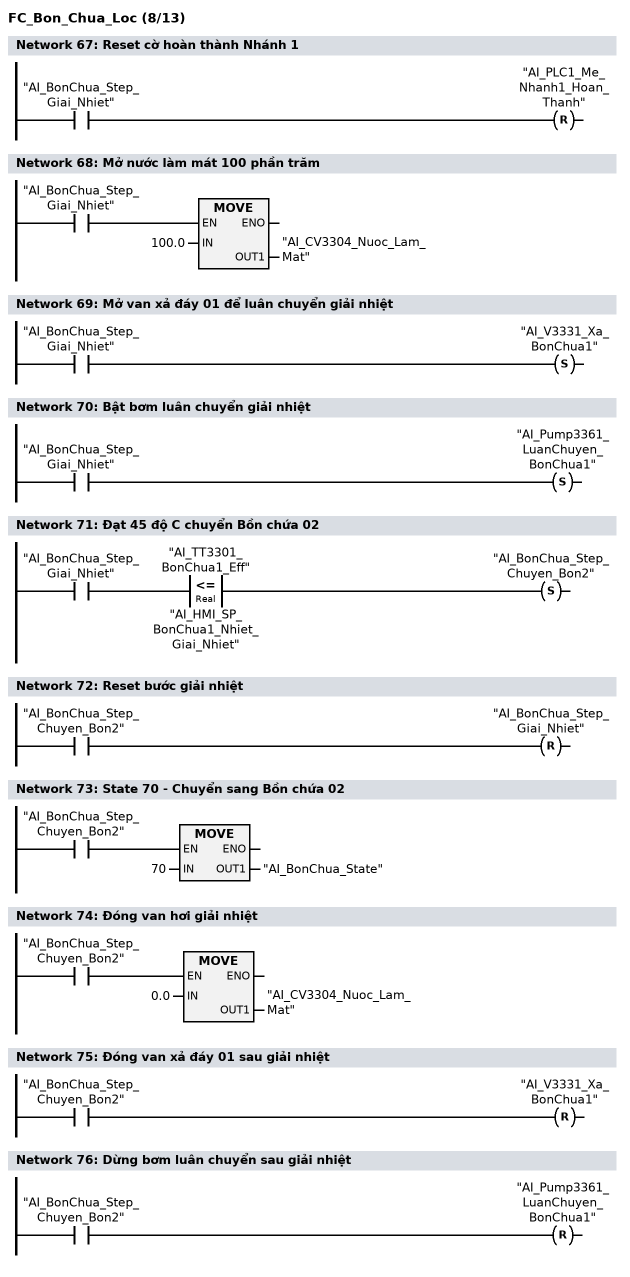
   RUNG wire#powerrail
      Contact( "AI_BonChua_Step_Giai_Nhiet" )
      R_Coil( "AI_PLC1_Me_Nhanh1_Hoan_Thanh" )
   END_RUNG
   // the same network as SCL:
   IF "AI_BonChua_Step_Giai_Nhiet" THEN "AI_PLC1_Me_Nhanh1_Hoan_Thanh" := FALSE; END_IF;
END_REGION

REGION Network 68: Mở nước làm mát 100 phần trăm
   RUNG wire#powerrail
      Contact( "AI_BonChua_Step_Giai_Nhiet" )
      { S7_GenerateENO := "TRUE" } Move(in := 100.0, out1 => "AI_CV3304_Nuoc_Lam_Mat")
   END_RUNG
   // the same network as SCL:
   IF "AI_BonChua_Step_Giai_Nhiet" THEN "AI_CV3304_Nuoc_Lam_Mat" := 100.0; END_IF;
END_REGION

REGION Network 69: Mở van xả đáy 01 để luân chuyển giải nhiệt
   RUNG wire#powerrail
      Contact( "AI_BonChua_Step_Giai_Nhiet" )
      S_Coil( "AI_V3331_Xa_BonChua1" )
   END_RUNG
   // the same network as SCL:
   IF "AI_BonChua_Step_Giai_Nhiet" THEN "AI_V3331_Xa_BonChua1" := TRUE; END_IF;
END_REGION

REGION Network 70: Bật bơm luân chuyển giải nhiệt
   RUNG wire#powerrail
      Contact( "AI_BonChua_Step_Giai_Nhiet" )
      S_Coil( "AI_Pump3361_LuanChuyen_BonChua1" )
   END_RUNG
   // the same network as SCL:
   IF "AI_BonChua_Step_Giai_Nhiet" THEN "AI_Pump3361_LuanChuyen_BonChua1" := TRUE; END_IF;
END_REGION

REGION Network 71: Đạt 45 độ C chuyển Bồn chứa 02
   RUNG wire#powerrail
      Contact( "AI_BonChua_Step_Giai_Nhiet" )
      { S7_Templates := "SrcType := Real" } LE_Contact(in1 := "AI_TT3301_BonChua1_Eff", in2 := "AI_HMI_SP_BonChua1_Nhiet_Giai_Nhiet")
      S_Coil( "AI_BonChua_Step_Chuyen_Bon2" )
   END_RUNG
   // the same network as SCL:
   IF "AI_BonChua_Step_Giai_Nhiet" AND ("AI_TT3301_BonChua1_Eff" <= "AI_HMI_SP_BonChua1_Nhiet_Giai_Nhiet") THEN
       "AI_BonChua_Step_Chuyen_Bon2" := TRUE;
   END_IF;
END_REGION

REGION Network 72: Reset bước giải nhiệt
   RUNG wire#powerrail
      Contact( "AI_BonChua_Step_Chuyen_Bon2" )
      R_Coil( "AI_BonChua_Step_Giai_Nhiet" )
   END_RUNG
   // the same network as SCL:
   IF "AI_BonChua_Step_Chuyen_Bon2" THEN "AI_BonChua_Step_Giai_Nhiet" := FALSE; END_IF;
END_REGION

REGION Network 73: State 70 - Chuyển sang Bồn chứa 02
   RUNG wire#powerrail
      Contact( "AI_BonChua_Step_Chuyen_Bon2" )
      { S7_GenerateENO := "TRUE" } Move(in := 70, out1 => "AI_BonChua_State")
   END_RUNG
   // the same network as SCL:
   IF "AI_BonChua_Step_Chuyen_Bon2" THEN "AI_BonChua_State" := 70; END_IF;
END_REGION

REGION Network 74: Đóng van hơi giải nhiệt
   RUNG wire#powerrail
      Contact( "AI_BonChua_Step_Chuyen_Bon2" )
      { S7_GenerateENO := "TRUE" } Move(in := 0.0, out1 => "AI_CV3304_Nuoc_Lam_Mat")
   END_RUNG
   // the same network as SCL:
   IF "AI_BonChua_Step_Chuyen_Bon2" THEN "AI_CV3304_Nuoc_Lam_Mat" := 0.0; END_IF;
END_REGION

REGION Network 75: Đóng van xả đáy 01 sau giải nhiệt
   RUNG wire#powerrail
      Contact( "AI_BonChua_Step_Chuyen_Bon2" )
      R_Coil( "AI_V3331_Xa_BonChua1" )
   END_RUNG
   // the same network as SCL:
   IF "AI_BonChua_Step_Chuyen_Bon2" THEN "AI_V3331_Xa_BonChua1" := FALSE; END_IF;
END_REGION

REGION Network 76: Dừng bơm luân chuyển sau giải nhiệt
   RUNG wire#powerrail
      Contact( "AI_BonChua_Step_Chuyen_Bon2" )
      R_Coil( "AI_Pump3361_LuanChuyen_BonChua1" )
   END_RUNG
   // the same network as SCL:
   IF "AI_BonChua_Step_Chuyen_Bon2" THEN "AI_Pump3361_LuanChuyen_BonChua1" := FALSE; END_IF;
END_REGION

REGION Network 77: Mở van xả đáy 02 để chuyển bồn
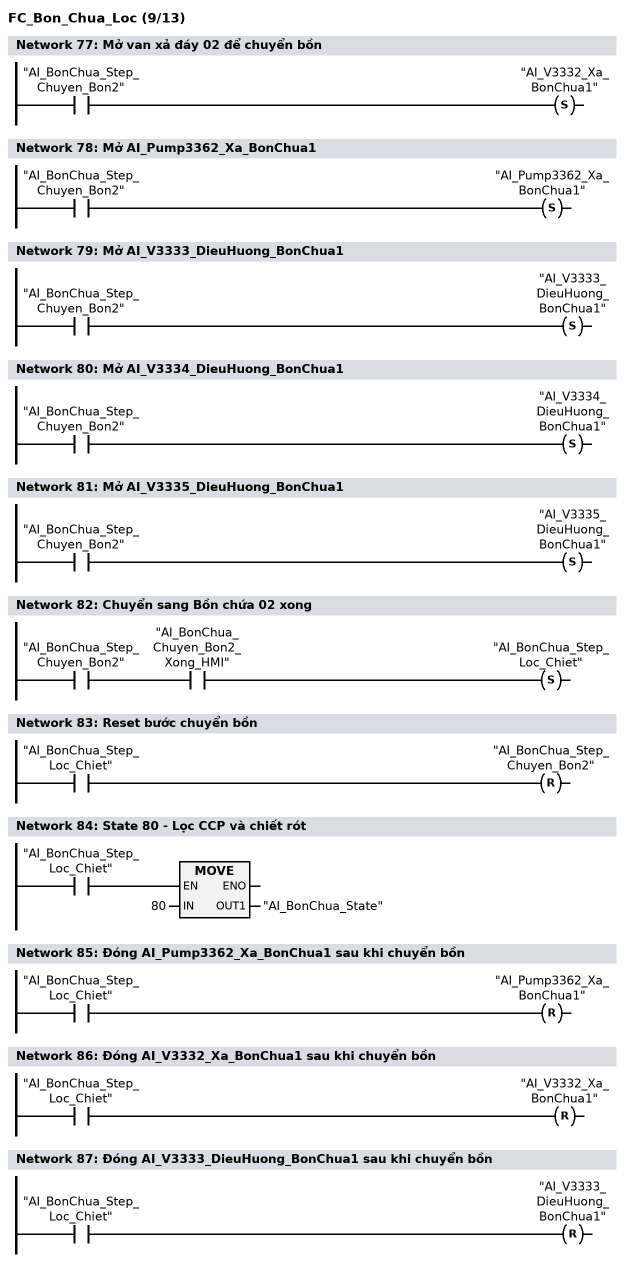
   RUNG wire#powerrail
      Contact( "AI_BonChua_Step_Chuyen_Bon2" )
      S_Coil( "AI_V3332_Xa_BonChua1" )
   END_RUNG
   // the same network as SCL:
   IF "AI_BonChua_Step_Chuyen_Bon2" THEN "AI_V3332_Xa_BonChua1" := TRUE; END_IF;
END_REGION

REGION Network 78: Mở AI_Pump3362_Xa_BonChua1
   RUNG wire#powerrail
      Contact( "AI_BonChua_Step_Chuyen_Bon2" )
      S_Coil( "AI_Pump3362_Xa_BonChua1" )
   END_RUNG
   // the same network as SCL:
   IF "AI_BonChua_Step_Chuyen_Bon2" THEN "AI_Pump3362_Xa_BonChua1" := TRUE; END_IF;
END_REGION

REGION Network 79: Mở AI_V3333_DieuHuong_BonChua1
   RUNG wire#powerrail
      Contact( "AI_BonChua_Step_Chuyen_Bon2" )
      S_Coil( "AI_V3333_DieuHuong_BonChua1" )
   END_RUNG
   // the same network as SCL:
   IF "AI_BonChua_Step_Chuyen_Bon2" THEN "AI_V3333_DieuHuong_BonChua1" := TRUE; END_IF;
END_REGION

REGION Network 80: Mở AI_V3334_DieuHuong_BonChua1
   RUNG wire#powerrail
      Contact( "AI_BonChua_Step_Chuyen_Bon2" )
      S_Coil( "AI_V3334_DieuHuong_BonChua1" )
   END_RUNG
   // the same network as SCL:
   IF "AI_BonChua_Step_Chuyen_Bon2" THEN "AI_V3334_DieuHuong_BonChua1" := TRUE; END_IF;
END_REGION

REGION Network 81: Mở AI_V3335_DieuHuong_BonChua1
   RUNG wire#powerrail
      Contact( "AI_BonChua_Step_Chuyen_Bon2" )
      S_Coil( "AI_V3335_DieuHuong_BonChua1" )
   END_RUNG
   // the same network as SCL:
   IF "AI_BonChua_Step_Chuyen_Bon2" THEN "AI_V3335_DieuHuong_BonChua1" := TRUE; END_IF;
END_REGION

REGION Network 82: Chuyển sang Bồn chứa 02 xong
   RUNG wire#powerrail
      Contact( "AI_BonChua_Step_Chuyen_Bon2" )
      Contact( "AI_BonChua_Chuyen_Bon2_Xong_HMI" )
      S_Coil( "AI_BonChua_Step_Loc_Chiet" )
   END_RUNG
   // the same network as SCL:
   IF "AI_BonChua_Step_Chuyen_Bon2" AND "AI_BonChua_Chuyen_Bon2_Xong_HMI" THEN
       "AI_BonChua_Step_Loc_Chiet" := TRUE;
   END_IF;
END_REGION

REGION Network 83: Reset bước chuyển bồn
   RUNG wire#powerrail
      Contact( "AI_BonChua_Step_Loc_Chiet" )
      R_Coil( "AI_BonChua_Step_Chuyen_Bon2" )
   END_RUNG
   // the same network as SCL:
   IF "AI_BonChua_Step_Loc_Chiet" THEN "AI_BonChua_Step_Chuyen_Bon2" := FALSE; END_IF;
END_REGION

REGION Network 84: State 80 - Lọc CCP và chiết rót
   RUNG wire#powerrail
      Contact( "AI_BonChua_Step_Loc_Chiet" )
      { S7_GenerateENO := "TRUE" } Move(in := 80, out1 => "AI_BonChua_State")
   END_RUNG
   // the same network as SCL:
   IF "AI_BonChua_Step_Loc_Chiet" THEN "AI_BonChua_State" := 80; END_IF;
END_REGION

REGION Network 85: Đóng AI_Pump3362_Xa_BonChua1 sau khi chuyển bồn
   RUNG wire#powerrail
      Contact( "AI_BonChua_Step_Loc_Chiet" )
      R_Coil( "AI_Pump3362_Xa_BonChua1" )
   END_RUNG
   // the same network as SCL:
   IF "AI_BonChua_Step_Loc_Chiet" THEN "AI_Pump3362_Xa_BonChua1" := FALSE; END_IF;
END_REGION

REGION Network 86: Đóng AI_V3332_Xa_BonChua1 sau khi chuyển bồn
   RUNG wire#powerrail
      Contact( "AI_BonChua_Step_Loc_Chiet" )
      R_Coil( "AI_V3332_Xa_BonChua1" )
   END_RUNG
   // the same network as SCL:
   IF "AI_BonChua_Step_Loc_Chiet" THEN "AI_V3332_Xa_BonChua1" := FALSE; END_IF;
END_REGION

REGION Network 87: Đóng AI_V3333_DieuHuong_BonChua1 sau khi chuyển bồn
   RUNG wire#powerrail
      Contact( "AI_BonChua_Step_Loc_Chiet" )
      R_Coil( "AI_V3333_DieuHuong_BonChua1" )
   END_RUNG
   // the same network as SCL:
   IF "AI_BonChua_Step_Loc_Chiet" THEN "AI_V3333_DieuHuong_BonChua1" := FALSE; END_IF;
END_REGION

REGION Network 88: Đóng AI_V3334_DieuHuong_BonChua1 sau khi chuyển bồn
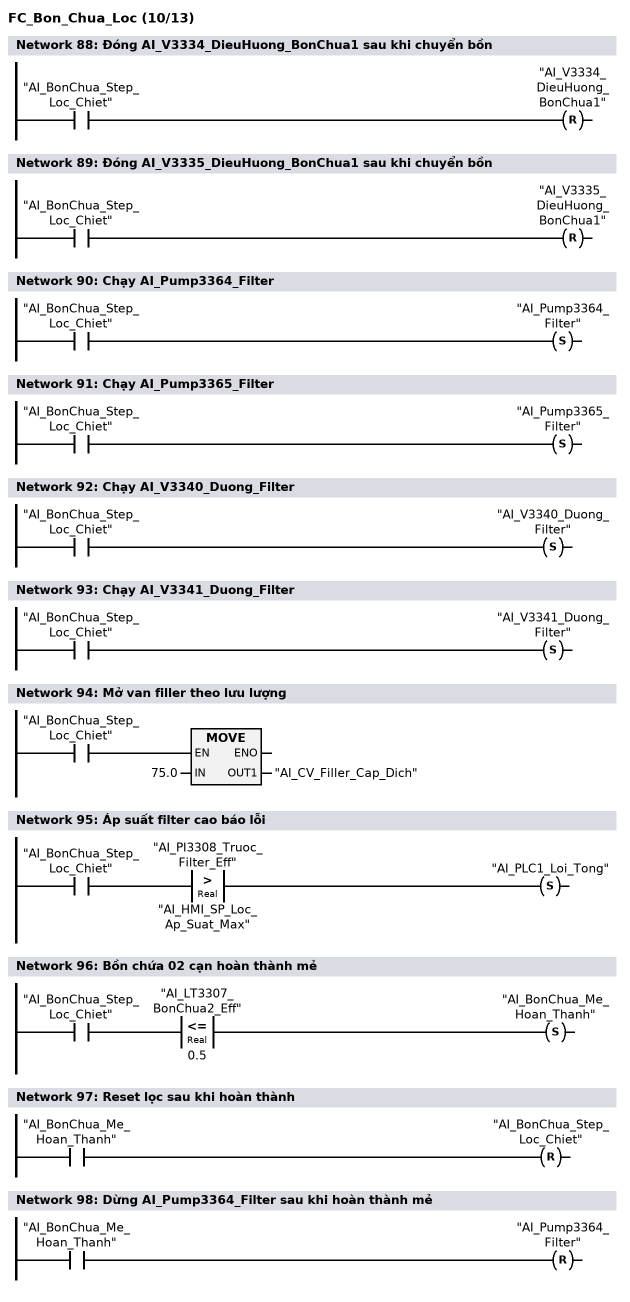
   RUNG wire#powerrail
      Contact( "AI_BonChua_Step_Loc_Chiet" )
      R_Coil( "AI_V3334_DieuHuong_BonChua1" )
   END_RUNG
   // the same network as SCL:
   IF "AI_BonChua_Step_Loc_Chiet" THEN "AI_V3334_DieuHuong_BonChua1" := FALSE; END_IF;
END_REGION

REGION Network 89: Đóng AI_V3335_DieuHuong_BonChua1 sau khi chuyển bồn
   RUNG wire#powerrail
      Contact( "AI_BonChua_Step_Loc_Chiet" )
      R_Coil( "AI_V3335_DieuHuong_BonChua1" )
   END_RUNG
   // the same network as SCL:
   IF "AI_BonChua_Step_Loc_Chiet" THEN "AI_V3335_DieuHuong_BonChua1" := FALSE; END_IF;
END_REGION

REGION Network 90: Chạy AI_Pump3364_Filter
   RUNG wire#powerrail
      Contact( "AI_BonChua_Step_Loc_Chiet" )
      S_Coil( "AI_Pump3364_Filter" )
   END_RUNG
   // the same network as SCL:
   IF "AI_BonChua_Step_Loc_Chiet" THEN "AI_Pump3364_Filter" := TRUE; END_IF;
END_REGION

REGION Network 91: Chạy AI_Pump3365_Filter
   RUNG wire#powerrail
      Contact( "AI_BonChua_Step_Loc_Chiet" )
      S_Coil( "AI_Pump3365_Filter" )
   END_RUNG
   // the same network as SCL:
   IF "AI_BonChua_Step_Loc_Chiet" THEN "AI_Pump3365_Filter" := TRUE; END_IF;
END_REGION

REGION Network 92: Chạy AI_V3340_Duong_Filter
   RUNG wire#powerrail
      Contact( "AI_BonChua_Step_Loc_Chiet" )
      S_Coil( "AI_V3340_Duong_Filter" )
   END_RUNG
   // the same network as SCL:
   IF "AI_BonChua_Step_Loc_Chiet" THEN "AI_V3340_Duong_Filter" := TRUE; END_IF;
END_REGION

REGION Network 93: Chạy AI_V3341_Duong_Filter
   RUNG wire#powerrail
      Contact( "AI_BonChua_Step_Loc_Chiet" )
      S_Coil( "AI_V3341_Duong_Filter" )
   END_RUNG
   // the same network as SCL:
   IF "AI_BonChua_Step_Loc_Chiet" THEN "AI_V3341_Duong_Filter" := TRUE; END_IF;
END_REGION

REGION Network 94: Mở van filler theo lưu lượng
   RUNG wire#powerrail
      Contact( "AI_BonChua_Step_Loc_Chiet" )
      { S7_GenerateENO := "TRUE" } Move(in := 75.0, out1 => "AI_CV_Filler_Cap_Dich")
   END_RUNG
   // the same network as SCL:
   IF "AI_BonChua_Step_Loc_Chiet" THEN "AI_CV_Filler_Cap_Dich" := 75.0; END_IF;
END_REGION

REGION Network 95: Áp suất filter cao báo lỗi
   RUNG wire#powerrail
      Contact( "AI_BonChua_Step_Loc_Chiet" )
      { S7_Templates := "SrcType := Real" } GT_Contact(in1 := "AI_PI3308_Truoc_Filter_Eff", in2 := "AI_HMI_SP_Loc_Ap_Suat_Max")
      S_Coil( "AI_PLC1_Loi_Tong" )
   END_RUNG
   // the same network as SCL:
   IF "AI_BonChua_Step_Loc_Chiet" AND ("AI_PI3308_Truoc_Filter_Eff" > "AI_HMI_SP_Loc_Ap_Suat_Max") THEN
       "AI_PLC1_Loi_Tong" := TRUE;
   END_IF;
END_REGION

REGION Network 96: Bồn chứa 02 cạn hoàn thành mẻ
   RUNG wire#powerrail
      Contact( "AI_BonChua_Step_Loc_Chiet" )
      { S7_Templates := "SrcType := Real" } LE_Contact(in1 := "AI_LT3307_BonChua2_Eff", in2 := 0.5)
      S_Coil( "AI_BonChua_Me_Hoan_Thanh" )
   END_RUNG
   // the same network as SCL:
   IF "AI_BonChua_Step_Loc_Chiet" AND ("AI_LT3307_BonChua2_Eff" <= 0.5) THEN
       "AI_BonChua_Me_Hoan_Thanh" := TRUE;
   END_IF;
END_REGION

REGION Network 97: Reset lọc sau khi hoàn thành
   RUNG wire#powerrail
      Contact( "AI_BonChua_Me_Hoan_Thanh" )
      R_Coil( "AI_BonChua_Step_Loc_Chiet" )
   END_RUNG
   // the same network as SCL:
   IF "AI_BonChua_Me_Hoan_Thanh" THEN "AI_BonChua_Step_Loc_Chiet" := FALSE; END_IF;
END_REGION

REGION Network 98: Dừng AI_Pump3364_Filter sau khi hoàn thành mẻ
   RUNG wire#powerrail
      Contact( "AI_BonChua_Me_Hoan_Thanh" )
      R_Coil( "AI_Pump3364_Filter" )
   END_RUNG
   // the same network as SCL:
   IF "AI_BonChua_Me_Hoan_Thanh" THEN "AI_Pump3364_Filter" := FALSE; END_IF;
END_REGION

REGION Network 99: Dừng AI_Pump3365_Filter sau khi hoàn thành mẻ
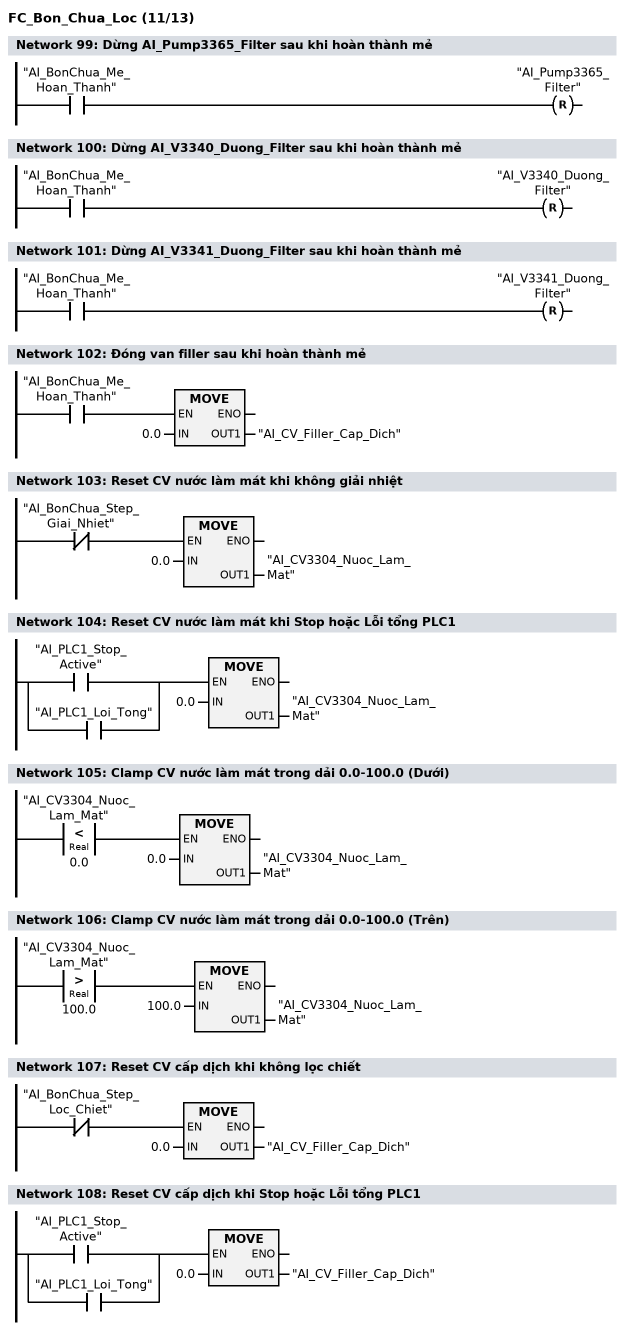
   RUNG wire#powerrail
      Contact( "AI_BonChua_Me_Hoan_Thanh" )
      R_Coil( "AI_Pump3365_Filter" )
   END_RUNG
   // the same network as SCL:
   IF "AI_BonChua_Me_Hoan_Thanh" THEN "AI_Pump3365_Filter" := FALSE; END_IF;
END_REGION

REGION Network 100: Dừng AI_V3340_Duong_Filter sau khi hoàn thành mẻ
   RUNG wire#powerrail
      Contact( "AI_BonChua_Me_Hoan_Thanh" )
      R_Coil( "AI_V3340_Duong_Filter" )
   END_RUNG
   // the same network as SCL:
   IF "AI_BonChua_Me_Hoan_Thanh" THEN "AI_V3340_Duong_Filter" := FALSE; END_IF;
END_REGION

REGION Network 101: Dừng AI_V3341_Duong_Filter sau khi hoàn thành mẻ
   RUNG wire#powerrail
      Contact( "AI_BonChua_Me_Hoan_Thanh" )
      R_Coil( "AI_V3341_Duong_Filter" )
   END_RUNG
   // the same network as SCL:
   IF "AI_BonChua_Me_Hoan_Thanh" THEN "AI_V3341_Duong_Filter" := FALSE; END_IF;
END_REGION

REGION Network 102: Đóng van filler sau khi hoàn thành mẻ
   RUNG wire#powerrail
      Contact( "AI_BonChua_Me_Hoan_Thanh" )
      { S7_GenerateENO := "TRUE" } Move(in := 0.0, out1 => "AI_CV_Filler_Cap_Dich")
   END_RUNG
   // the same network as SCL:
   IF "AI_BonChua_Me_Hoan_Thanh" THEN "AI_CV_Filler_Cap_Dich" := 0.0; END_IF;
END_REGION

REGION Network 103: Reset CV nước làm mát khi không giải nhiệt
   RUNG wire#powerrail
      I_Contact( "AI_BonChua_Step_Giai_Nhiet" )
      { S7_GenerateENO := "TRUE" } Move(in := 0.0, out1 => "AI_CV3304_Nuoc_Lam_Mat")
   END_RUNG
   // the same network as SCL:
   IF NOT "AI_BonChua_Step_Giai_Nhiet" THEN "AI_CV3304_Nuoc_Lam_Mat" := 0.0; END_IF;
END_REGION

REGION Network 104: Reset CV nước làm mát khi Stop hoặc Lỗi tổng PLC1
   RUNG wire#powerrail
      Contact( "AI_PLC1_Stop_Active" )
      wire#w1
      { S7_GenerateENO := "TRUE" } Move(in := 0.0, out1 => "AI_CV3304_Nuoc_Lam_Mat")
   END_RUNG
   RUNG wire#powerrail
      Contact( "AI_PLC1_Loi_Tong" )
   END_RUNG wire#w1
   // the same network as SCL:
   IF "AI_PLC1_Stop_Active" OR "AI_PLC1_Loi_Tong" THEN "AI_CV3304_Nuoc_Lam_Mat" := 0.0; END_IF;
END_REGION

REGION Network 105: Clamp CV nước làm mát trong dải 0.0-100.0 (Dưới)
   RUNG wire#powerrail
      { S7_Templates := "SrcType := Real" } LT_Contact(in1 := "AI_CV3304_Nuoc_Lam_Mat", in2 := 0.0)
      { S7_GenerateENO := "TRUE" } Move(in := 0.0, out1 => "AI_CV3304_Nuoc_Lam_Mat")
   END_RUNG
   // the same network as SCL:
   IF "AI_CV3304_Nuoc_Lam_Mat" < 0.0 THEN "AI_CV3304_Nuoc_Lam_Mat" := 0.0; END_IF;
END_REGION

REGION Network 106: Clamp CV nước làm mát trong dải 0.0-100.0 (Trên)
   RUNG wire#powerrail
      { S7_Templates := "SrcType := Real" } GT_Contact(in1 := "AI_CV3304_Nuoc_Lam_Mat", in2 := 100.0)
      { S7_GenerateENO := "TRUE" } Move(in := 100.0, out1 => "AI_CV3304_Nuoc_Lam_Mat")
   END_RUNG
   // the same network as SCL:
   IF "AI_CV3304_Nuoc_Lam_Mat" > 100.0 THEN "AI_CV3304_Nuoc_Lam_Mat" := 100.0; END_IF;
END_REGION

REGION Network 107: Reset CV cấp dịch khi không lọc chiết
   RUNG wire#powerrail
      I_Contact( "AI_BonChua_Step_Loc_Chiet" )
      { S7_GenerateENO := "TRUE" } Move(in := 0.0, out1 => "AI_CV_Filler_Cap_Dich")
   END_RUNG
   // the same network as SCL:
   IF NOT "AI_BonChua_Step_Loc_Chiet" THEN "AI_CV_Filler_Cap_Dich" := 0.0; END_IF;
END_REGION

REGION Network 108: Reset CV cấp dịch khi Stop hoặc Lỗi tổng PLC1
   RUNG wire#powerrail
      Contact( "AI_PLC1_Stop_Active" )
      wire#w1
      { S7_GenerateENO := "TRUE" } Move(in := 0.0, out1 => "AI_CV_Filler_Cap_Dich")
   END_RUNG
   RUNG wire#powerrail
      Contact( "AI_PLC1_Loi_Tong" )
   END_RUNG wire#w1
   // the same network as SCL:
   IF "AI_PLC1_Stop_Active" OR "AI_PLC1_Loi_Tong" THEN "AI_CV_Filler_Cap_Dich" := 0.0; END_IF;
END_REGION

REGION Network 109: Clamp CV cấp dịch trong dải 0.0-100.0 (Dưới)
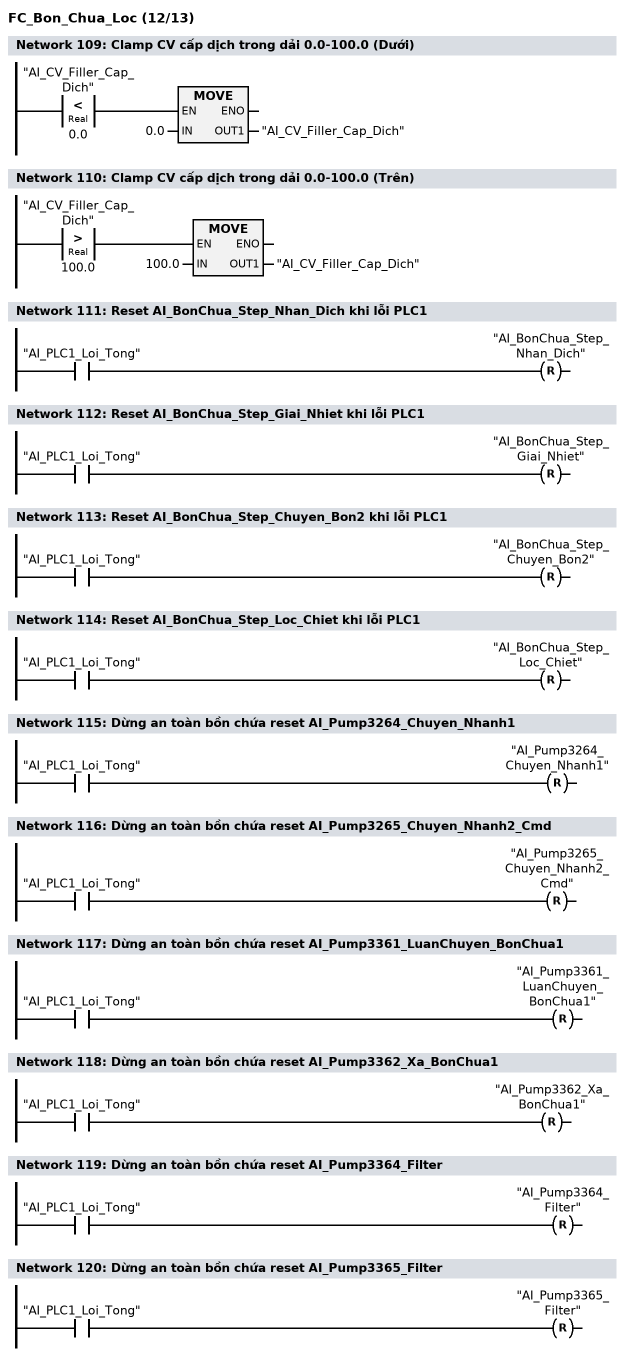
   RUNG wire#powerrail
      { S7_Templates := "SrcType := Real" } LT_Contact(in1 := "AI_CV_Filler_Cap_Dich", in2 := 0.0)
      { S7_GenerateENO := "TRUE" } Move(in := 0.0, out1 => "AI_CV_Filler_Cap_Dich")
   END_RUNG
   // the same network as SCL:
   IF "AI_CV_Filler_Cap_Dich" < 0.0 THEN "AI_CV_Filler_Cap_Dich" := 0.0; END_IF;
END_REGION

REGION Network 110: Clamp CV cấp dịch trong dải 0.0-100.0 (Trên)
   RUNG wire#powerrail
      { S7_Templates := "SrcType := Real" } GT_Contact(in1 := "AI_CV_Filler_Cap_Dich", in2 := 100.0)
      { S7_GenerateENO := "TRUE" } Move(in := 100.0, out1 => "AI_CV_Filler_Cap_Dich")
   END_RUNG
   // the same network as SCL:
   IF "AI_CV_Filler_Cap_Dich" > 100.0 THEN "AI_CV_Filler_Cap_Dich" := 100.0; END_IF;
END_REGION

REGION Network 111: Reset AI_BonChua_Step_Nhan_Dich khi lỗi PLC1
   RUNG wire#powerrail
      Contact( "AI_PLC1_Loi_Tong" )
      R_Coil( "AI_BonChua_Step_Nhan_Dich" )
   END_RUNG
   // the same network as SCL:
   IF "AI_PLC1_Loi_Tong" THEN "AI_BonChua_Step_Nhan_Dich" := FALSE; END_IF;
END_REGION

REGION Network 112: Reset AI_BonChua_Step_Giai_Nhiet khi lỗi PLC1
   RUNG wire#powerrail
      Contact( "AI_PLC1_Loi_Tong" )
      R_Coil( "AI_BonChua_Step_Giai_Nhiet" )
   END_RUNG
   // the same network as SCL:
   IF "AI_PLC1_Loi_Tong" THEN "AI_BonChua_Step_Giai_Nhiet" := FALSE; END_IF;
END_REGION

REGION Network 113: Reset AI_BonChua_Step_Chuyen_Bon2 khi lỗi PLC1
   RUNG wire#powerrail
      Contact( "AI_PLC1_Loi_Tong" )
      R_Coil( "AI_BonChua_Step_Chuyen_Bon2" )
   END_RUNG
   // the same network as SCL:
   IF "AI_PLC1_Loi_Tong" THEN "AI_BonChua_Step_Chuyen_Bon2" := FALSE; END_IF;
END_REGION

REGION Network 114: Reset AI_BonChua_Step_Loc_Chiet khi lỗi PLC1
   RUNG wire#powerrail
      Contact( "AI_PLC1_Loi_Tong" )
      R_Coil( "AI_BonChua_Step_Loc_Chiet" )
   END_RUNG
   // the same network as SCL:
   IF "AI_PLC1_Loi_Tong" THEN "AI_BonChua_Step_Loc_Chiet" := FALSE; END_IF;
END_REGION

REGION Network 115: Dừng an toàn bồn chứa reset AI_Pump3264_Chuyen_Nhanh1
   RUNG wire#powerrail
      Contact( "AI_PLC1_Loi_Tong" )
      R_Coil( "AI_Pump3264_Chuyen_Nhanh1" )
   END_RUNG
   // the same network as SCL:
   IF "AI_PLC1_Loi_Tong" THEN "AI_Pump3264_Chuyen_Nhanh1" := FALSE; END_IF;
END_REGION

REGION Network 116: Dừng an toàn bồn chứa reset AI_Pump3265_Chuyen_Nhanh2_Cmd
   RUNG wire#powerrail
      Contact( "AI_PLC1_Loi_Tong" )
      R_Coil( "AI_Pump3265_Chuyen_Nhanh2_Cmd" )
   END_RUNG
   // the same network as SCL:
   IF "AI_PLC1_Loi_Tong" THEN "AI_Pump3265_Chuyen_Nhanh2_Cmd" := FALSE; END_IF;
END_REGION

REGION Network 117: Dừng an toàn bồn chứa reset AI_Pump3361_LuanChuyen_BonChua1
   RUNG wire#powerrail
      Contact( "AI_PLC1_Loi_Tong" )
      R_Coil( "AI_Pump3361_LuanChuyen_BonChua1" )
   END_RUNG
   // the same network as SCL:
   IF "AI_PLC1_Loi_Tong" THEN "AI_Pump3361_LuanChuyen_BonChua1" := FALSE; END_IF;
END_REGION

REGION Network 118: Dừng an toàn bồn chứa reset AI_Pump3362_Xa_BonChua1
   RUNG wire#powerrail
      Contact( "AI_PLC1_Loi_Tong" )
      R_Coil( "AI_Pump3362_Xa_BonChua1" )
   END_RUNG
   // the same network as SCL:
   IF "AI_PLC1_Loi_Tong" THEN "AI_Pump3362_Xa_BonChua1" := FALSE; END_IF;
END_REGION

REGION Network 119: Dừng an toàn bồn chứa reset AI_Pump3364_Filter
   RUNG wire#powerrail
      Contact( "AI_PLC1_Loi_Tong" )
      R_Coil( "AI_Pump3364_Filter" )
   END_RUNG
   // the same network as SCL:
   IF "AI_PLC1_Loi_Tong" THEN "AI_Pump3364_Filter" := FALSE; END_IF;
END_REGION

REGION Network 120: Dừng an toàn bồn chứa reset AI_Pump3365_Filter
   RUNG wire#powerrail
      Contact( "AI_PLC1_Loi_Tong" )
      R_Coil( "AI_Pump3365_Filter" )
   END_RUNG
   // the same network as SCL:
   IF "AI_PLC1_Loi_Tong" THEN "AI_Pump3365_Filter" := FALSE; END_IF;
END_REGION

REGION Network 121: Dừng an toàn bồn chứa reset AI_V3331_Xa_BonChua1
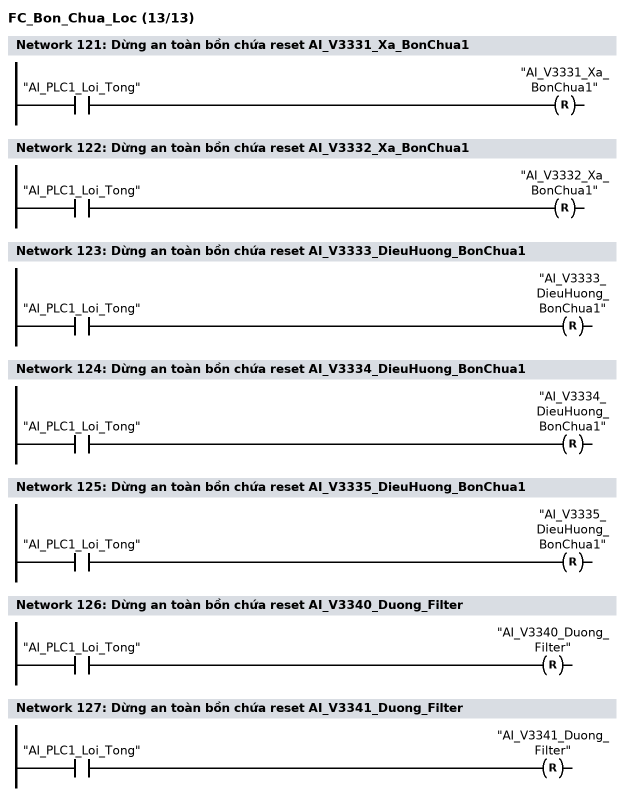
   RUNG wire#powerrail
      Contact( "AI_PLC1_Loi_Tong" )
      R_Coil( "AI_V3331_Xa_BonChua1" )
   END_RUNG
   // the same network as SCL:
   IF "AI_PLC1_Loi_Tong" THEN "AI_V3331_Xa_BonChua1" := FALSE; END_IF;
END_REGION

REGION Network 122: Dừng an toàn bồn chứa reset AI_V3332_Xa_BonChua1
   RUNG wire#powerrail
      Contact( "AI_PLC1_Loi_Tong" )
      R_Coil( "AI_V3332_Xa_BonChua1" )
   END_RUNG
   // the same network as SCL:
   IF "AI_PLC1_Loi_Tong" THEN "AI_V3332_Xa_BonChua1" := FALSE; END_IF;
END_REGION

REGION Network 123: Dừng an toàn bồn chứa reset AI_V3333_DieuHuong_BonChua1
   RUNG wire#powerrail
      Contact( "AI_PLC1_Loi_Tong" )
      R_Coil( "AI_V3333_DieuHuong_BonChua1" )
   END_RUNG
   // the same network as SCL:
   IF "AI_PLC1_Loi_Tong" THEN "AI_V3333_DieuHuong_BonChua1" := FALSE; END_IF;
END_REGION

REGION Network 124: Dừng an toàn bồn chứa reset AI_V3334_DieuHuong_BonChua1
   RUNG wire#powerrail
      Contact( "AI_PLC1_Loi_Tong" )
      R_Coil( "AI_V3334_DieuHuong_BonChua1" )
   END_RUNG
   // the same network as SCL:
   IF "AI_PLC1_Loi_Tong" THEN "AI_V3334_DieuHuong_BonChua1" := FALSE; END_IF;
END_REGION

REGION Network 125: Dừng an toàn bồn chứa reset AI_V3335_DieuHuong_BonChua1
   RUNG wire#powerrail
      Contact( "AI_PLC1_Loi_Tong" )
      R_Coil( "AI_V3335_DieuHuong_BonChua1" )
   END_RUNG
   // the same network as SCL:
   IF "AI_PLC1_Loi_Tong" THEN "AI_V3335_DieuHuong_BonChua1" := FALSE; END_IF;
END_REGION

REGION Network 126: Dừng an toàn bồn chứa reset AI_V3340_Duong_Filter
   RUNG wire#powerrail
      Contact( "AI_PLC1_Loi_Tong" )
      R_Coil( "AI_V3340_Duong_Filter" )
   END_RUNG
   // the same network as SCL:
   IF "AI_PLC1_Loi_Tong" THEN "AI_V3340_Duong_Filter" := FALSE; END_IF;
END_REGION

REGION Network 127: Dừng an toàn bồn chứa reset AI_V3341_Duong_Filter
   RUNG wire#powerrail
      Contact( "AI_PLC1_Loi_Tong" )
      R_Coil( "AI_V3341_Duong_Filter" )
   END_RUNG
   // the same network as SCL:
   IF "AI_PLC1_Loi_Tong" THEN "AI_V3341_Duong_Filter" := FALSE; END_IF;
END_REGION
END_FUNCTION
